Staubli VAL3: stop.pgx

program stop()
begin
  //
  call IO:CloseAll()
  taskKill("light")
  PublicData:libSave()
end
